FUNCTION F_ToANY : __SYSTEM.AnyType
VAR_INPUT
	Input: ANY;
END_VAR
VAR
END_VAR

F_ToANY:= Input;

END_FUNCTION

(* stored: POU F_ToANY: Id 230d28cd-b685-4ae7-b48f-56431857e8ce, SpecialFunc None *)
